SUBAPPLICATION AUDI_AUI_MUX_6_VAL (* 6-Wege-Multiplexer fuer AUDI-Werte mit 6 internen initval_AUDI und AUI_MUX_6 / AUDI_AUI_MUX_6. Schaltet per Event-Input (EI1..EI6) zwischen val1..val6 um. *)
  (* Standard: 61499-2; Description: Copyright (c) 2026 Meisterschulen am Ostbahnhof This program and the accompanying materials are made available under the terms of the Eclipse Public License 2.0 which is available at https://www.eclipse.org/legal/epl-2.0/ SPDX-License-Identifier: EPL-2.0 *)
  (* Version 1.0, 2026-09-10, Franz Höpfinger, Meisterschulen am Ostbahnhof, 6-fach Variante von AUDI_AUI_MUX_3_VAL *)
  PACKAGE MyLib::sys;
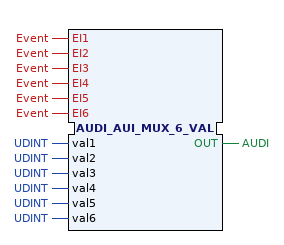
  EVENT_INPUT
    EI1; (* Event zur Auswahl von val1 *)
    EI2; (* Event zur Auswahl von val2 *)
    EI3; (* Event zur Auswahl von val3 *)
    EI4; (* Event zur Auswahl von val4 *)
    EI5; (* Event zur Auswahl von val5 *)
    EI6; (* Event zur Auswahl von val6 *)
  END_EVENT
  VAR_INPUT
    val1 : UDINT; (* Initialer Ausgabewert bei EI1 *)
    val2 : UDINT; (* Initialer Ausgabewert bei EI2 *)
    val3 : UDINT; (* Initialer Ausgabewert bei EI3 *)
    val4 : UDINT; (* Initialer Ausgabewert bei EI4 *)
    val5 : UDINT; (* Initialer Ausgabewert bei EI5 *)
    val6 : UDINT; (* Initialer Ausgabewert bei EI6 *)
  END_VAR
  PLUGS
    OUT : adapter::types::unidirectional::AUDI; (* Ausgewaehlter AUDI-Adapter Output *)
  END_PLUGS
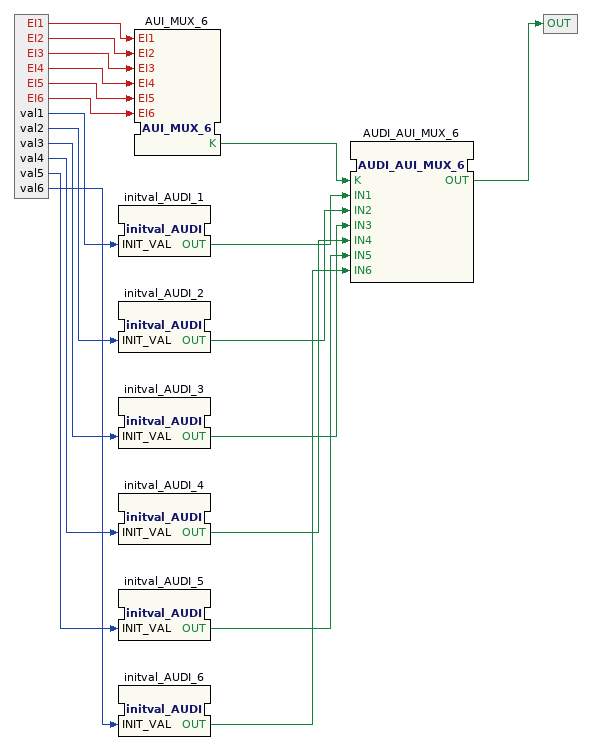
  FBS
    AUI_MUX_6 : adapter::events::unidirectional::AUI_MUX_6;
    AUDI_AUI_MUX_6 : adapter::selection::unidirectional::AUDI_AUI_MUX_6;
    initval_AUDI_1 : adapter::types::unidirectional::AUDI::initval::initval_AUDI;
    initval_AUDI_2 : adapter::types::unidirectional::AUDI::initval::initval_AUDI;
    initval_AUDI_3 : adapter::types::unidirectional::AUDI::initval::initval_AUDI;
    initval_AUDI_4 : adapter::types::unidirectional::AUDI::initval::initval_AUDI;
    initval_AUDI_5 : adapter::types::unidirectional::AUDI::initval::initval_AUDI;
    initval_AUDI_6 : adapter::types::unidirectional::AUDI::initval::initval_AUDI;
  END_FBS
  EVENT_CONNECTIONS
    EI1 TO AUI_MUX_6.EI1;
    EI2 TO AUI_MUX_6.EI2;
    EI3 TO AUI_MUX_6.EI3;
    EI4 TO AUI_MUX_6.EI4;
    EI5 TO AUI_MUX_6.EI5;
    EI6 TO AUI_MUX_6.EI6;
  END_CONNECTIONS
  DATA_CONNECTIONS
    val1 TO initval_AUDI_1.INIT_VAL;
    val2 TO initval_AUDI_2.INIT_VAL;
    val3 TO initval_AUDI_3.INIT_VAL;
    val4 TO initval_AUDI_4.INIT_VAL;
    val5 TO initval_AUDI_5.INIT_VAL;
    val6 TO initval_AUDI_6.INIT_VAL;
  END_CONNECTIONS
  ADAPTER_CONNECTIONS
    AUI_MUX_6.K TO AUDI_AUI_MUX_6.K;
    initval_AUDI_1.OUT TO AUDI_AUI_MUX_6.IN1;
    initval_AUDI_2.OUT TO AUDI_AUI_MUX_6.IN2;
    initval_AUDI_3.OUT TO AUDI_AUI_MUX_6.IN3;
    initval_AUDI_4.OUT TO AUDI_AUI_MUX_6.IN4;
    initval_AUDI_5.OUT TO AUDI_AUI_MUX_6.IN5;
    initval_AUDI_6.OUT TO AUDI_AUI_MUX_6.IN6;
    AUDI_AUI_MUX_6.OUT TO OUT;
  END_CONNECTIONS
END_SUBAPPLICATION
